FUNCTION_BLOCK SampleContext EXTENDS TcoCore.TcoContext
VAR
	_sampleComponent : SampleComponent(THIS^, TcoCore.NO.Structure);
END_VAR

(*~
	<docu>
		<summary>
			Main method of the TcoContext. This is the entry point of any control logic that belongs to this context. 
			The call of this method is ensured by calling the <c>InstanceName.Run()</c> method, and it must not be called explicitly.
			This method is abstract, and it must be overridden in derived block.
		</summary>
	</docu>
~*)
METHOD PROTECTED  Main
_sampleComponent.Service();
_sampleComponent();
END_METHOD

END_FUNCTION_BLOCK

(* stored: Version 1.1.0.1, ProductVersion 3.1.4024.9
   POU SampleContext: Id {17b40f53-8ddf-02a7-0c48-23be770b6c32}, SpecialFunc None
   Method Main: Id {b16c1f30-7567-0482-3818-51b562bd8312} *)
